// TIA Portal V20 export
DATA_BLOCK "OPMODE01_OPEN_DOOR_IDB"   // DB88
// stored: AssignedProDiagFB OPMODE01_PD, InstanceOfName COND_PD_FB, InstanceOfType FB
"COND_PD_FB"
   // VAR_INPUT
   //    PD_TEXT { ExternalAccessible := 'False'; ExternalVisible := 'False'; ExternalWritable := 'False'} : WString[24];
   //    COND_NUMBER { ExternalAccessible := 'False'; ExternalVisible := 'False'; ExternalWritable := 'False'} : Int;
   //    COND_LOGIC { ExternalAccessible := 'False'; ExternalVisible := 'False'; ExternalWritable := 'False'} : Bool;
   //    CODE_VIEW_ENABLE { ExternalAccessible := 'False'; ExternalVisible := 'False'; ExternalWritable := 'False'} : Bool;
   // END_VAR
   // VAR_OUTPUT
   //    COND_OK { ExternalAccessible := 'False'; ExternalVisible := 'False'; ExternalWritable := 'False'} : Bool;
   // END_VAR
   // VAR_IN_OUT
   //    "IF" : "COND_PD_UDT";
   // END_VAR
   // VAR
   //    Code_View_Enabled { ExternalAccessible := 'False'; ExternalVisible := 'False'; ExternalWritable := 'False'} : Bool;
   // END_VAR
BEGIN
END_DATA_BLOCK
